// TwinCAT 3 PLC project PLC
// ProgramVersion: 3.1.4023.0
// libraries:
//   Tc2_ModbusRTU, * (Beckhoff Automation GmbH)
//   Tc2_Standard, * (Beckhoff Automation GmbH)
//   Tc2_System, * (Beckhoff Automation GmbH)
//   Tc2_Utilities, * (Beckhoff Automation GmbH)
//   Tc3_Module, * (Beckhoff Automation GmbH)
//   VisuSymbols,3.5.10.0,System
// project tree:
//   / GlobalTextList.TcGTLO, PlcTask.TcTTO, VISU_TASK.TcTTO
//   POUs/ FB_CalculateAI.TcPOU, FB_Modbus.TcPOU, FB_ModbusMaster.TcPOU, FB_ModbusSlave.TcPOU, FB_PM2200.TcPOU, FB_TDS3000.TcPOU, FB_TDS4339.TcPOU, I_ModbusSlave.TcIO (not stored), MAIN.TcPOU, U_Word2Real.TcDUT
//   VISUs/ Visualization.TcVIS, VisualizationManager.TcVMO (not stored)
// real-time tasks:
//   TASK PlcTask: cycle T#10ms, priority 20, ADS port 350
//   TASK VISU_TASK: cycle T#200000us, priority 30, ADS port 351
// I/O:
//   DEVICE Device 1 (EtherCAT) (disabled), AmsNetId 10.20.253.152.2.1
//     Term 1 (EK1200) [EK1200-5000 EtherCAT Power supply (2A E-Bus)]
//       Term 16 (EL1859) [EL1859 8Ch. Dig. Input 24V, 3ms, 8Ch. Dig. Output 24V, 0.5A]
//       Term 17 (EL1859) [EL1859 8Ch. Dig. Input 24V, 3ms, 8Ch. Dig. Output 24V, 0.5A]
//       Term 2 (EL1819) [EL1819 16Ch. Dig. Input 24V, 10µs]
//       Term 3 (EL1819) [EL1819 16Ch. Dig. Input 24V, 10µs]
//       Term 4 (EL1819) [EL1819 16Ch. Dig. Input 24V, 10µs]
//       Term 5 (EL1819) [EL1819 16Ch. Dig. Input 24V, 10µs]
//       Term 6 (EL1819) [EL1819 16Ch. Dig. Input 24V, 10µs]
//       Term 7 (EL1819) [EL1819 16Ch. Dig. Input 24V, 10µs]
//       Term 8 (EL1819) [EL1819 16Ch. Dig. Input 24V, 10µs]
//       Term 9 (EL2809) [EL2809 16Ch. Dig. Output 24V, 0.5A]
//       Term 10 (EL2809) [EL2809 16Ch. Dig. Output 24V, 0.5A]
//       Term 11 (EL3058) [EL3058 8Ch. Ana. Input 4-20mA]
//       Term 12 (EL6021) [EL6021 Interface (RS422/485)]
//       Term 30 (EL6021) [EL6021 Interface (RS422/485)]
//       Term 14 (EL9011) [EL9011 End Terminal]
//   DEVICE Device 2 (EtherCAT) (disabled), AmsNetId 192.168.56.1.3.1
//     Term 13 (EK1100) [EK1100 EtherCAT Coupler (2A E-Bus)]
//       Term 15 (EL6021) [EL6021 Interface (RS422/485)]
//   DEVICE Device 3 (COM Port)
// variable links:
//   PLC/PLC Instance <-> Device 1 (EtherCAT)/Term 1 (EK1200)/Term 10 (EL2809)
//     PlcTask Outputs/MAIN.bDO21 <-> Channel 1/Output
//     PlcTask Outputs/MAIN.bDO210 <-> Channel 10/Output
//     PlcTask Outputs/MAIN.bDO211 <-> Channel 11/Output
//     PlcTask Outputs/MAIN.bDO212 <-> Channel 12/Output
//     PlcTask Outputs/MAIN.bDO213 <-> Channel 13/Output
//     PlcTask Outputs/MAIN.bDO214 <-> Channel 14/Output
//     PlcTask Outputs/MAIN.bDO215 <-> Channel 15/Output
//     PlcTask Outputs/MAIN.bDO216 <-> Channel 16/Output
//     PlcTask Outputs/MAIN.bDO22 <-> Channel 2/Output
//     PlcTask Outputs/MAIN.bDO23 <-> Channel 3/Output
//     PlcTask Outputs/MAIN.bDO24 <-> Channel 4/Output
//     PlcTask Outputs/MAIN.bDO25 <-> Channel 5/Output
//     PlcTask Outputs/MAIN.bDO26 <-> Channel 6/Output
//     PlcTask Outputs/MAIN.bDO27 <-> Channel 7/Output
//     PlcTask Outputs/MAIN.bDO28 <-> Channel 8/Output
//     PlcTask Outputs/MAIN.bDO29 <-> Channel 9/Output
//   PLC/PLC Instance <-> Device 1 (EtherCAT)/Term 1 (EK1200)/Term 11 (EL3058)
//     PlcTask Inputs/MAIN.AI_DraftT1Case_Pressure <-> AI Standard Channel 7/Value
//     PlcTask Inputs/MAIN.AI_DraftT2Case_Voltage <-> AI Standard Channel 8/Value
//     PlcTask Inputs/MAIN.AI_Excitatiob_Current <-> AI Standard Channel 4/Value
//     PlcTask Inputs/MAIN.AI_Excitatiob_Voltage <-> AI Standard Channel 3/Value
//     PlcTask Inputs/MAIN.AI_GovernorBlOilade_Pressure <-> AI Standard Channel 2/Value
//     PlcTask Inputs/MAIN.AI_GovernorGuideVaneOil_Preesure <-> AI Standard Channel 1/Value
//     PlcTask Inputs/MAIN.AI_HeadCase_Pressure <-> AI Standard Channel 6/Value
//     PlcTask Inputs/MAIN.AI_SpiralCase_Pressure <-> AI Standard Channel 5/Value
//   PLC/PLC Instance <-> Device 1 (EtherCAT)/Term 1 (EK1200)/Term 9 (EL2809)
//     PlcTask Outputs/MAIN.bDO11 <-> Channel 1/Output
//     PlcTask Outputs/MAIN.bDO110 <-> Channel 10/Output
//     PlcTask Outputs/MAIN.bDO111 <-> Channel 11/Output
//     PlcTask Outputs/MAIN.bDO112 <-> Channel 12/Output
//     PlcTask Outputs/MAIN.bDO113 <-> Channel 13/Output
//     PlcTask Outputs/MAIN.bDO114 <-> Channel 14/Output
//     PlcTask Outputs/MAIN.bDO115 <-> Channel 15/Output
//     PlcTask Outputs/MAIN.bDO116 <-> Channel 16/Output
//     PlcTask Outputs/MAIN.bDO12 <-> Channel 2/Output
//     PlcTask Outputs/MAIN.bDO13 <-> Channel 3/Output
//     PlcTask Outputs/MAIN.bDO14 <-> Channel 4/Output
//     PlcTask Outputs/MAIN.bDO15 <-> Channel 5/Output
//     PlcTask Outputs/MAIN.bDO16 <-> Channel 6/Output
//     PlcTask Outputs/MAIN.bDO17 <-> Channel 7/Output
//     PlcTask Outputs/MAIN.bDO18 <-> Channel 8/Output
//     PlcTask Outputs/MAIN.bDO19 <-> Channel 9/Output

CONFIGURATION PLC
    RESOURCE PLC ON TwinCAT3
        TASK PlcTask(INTERVAL := T#10ms, PRIORITY := 20);
        TASK VISU_TASK(INTERVAL := T#200000us, PRIORITY := 30);
        PROGRAM MAIN WITH PlcTask : MAIN;
        PROGRAM VisuElems_Visu_Prg WITH VISU_TASK : VisuElems.Visu_Prg;
    END_RESOURCE
END_CONFIGURATION

// ---- POUs/U_Word2Real.TcDUT
TYPE U_Word2Real :
UNION
	iWord: ARRAY [0..1] OF WORD;
	rReal: REAL;
END_UNION
END_TYPE

// ---- POUs/MAIN.TcPOU
PROGRAM MAIN
VAR
	bDO11 AT %Q* :BOOL;
	bDO12 AT %Q*	:BOOL;
	bDO13 AT %Q*	:BOOL;
	bDO14 AT %Q*	:BOOL;
	bDO15 AT %Q*	:BOOL;
	bDO16 AT %Q*	:BOOL;
	bDO17 AT %Q*	:BOOL;
	bDO18 AT %Q*	:BOOL;
	bDO19 AT %Q*	:BOOL;
	bDO110 AT %Q* :BOOL;
	bDO111 AT %Q* :BOOL;
	bDO112 AT %Q* :BOOL;
	bDO113 AT %Q* :BOOL;
	bDO114 AT %Q* :BOOL;
	bDO115 AT %Q* :BOOL;
	bDO116 AT %Q* :BOOL;
		
	bDO21 AT %Q* :BOOL;
	bDO22 AT %Q*:BOOL;
	bDO23 AT %Q*:BOOL;
	bDO24 AT %Q*:BOOL;
	bDO25 AT %Q*:BOOL;
	bDO26 AT %Q*:BOOL;
	bDO27 AT %Q*:BOOL;
	bDO28 AT %Q*:BOOL;
	bDO29 AT %Q*:BOOL;
	bDO210 AT %Q* :BOOL;
	bDO211 AT %Q* :BOOL;
	bDO212 AT %Q* :BOOL;
	bDO213 AT %Q* :BOOL;
	bDO214 AT %Q* :BOOL;
	bDO215 AT %Q* :BOOL;
	bDO216 AT %Q* :BOOL;
	
	AI_GovernorGuideVaneOil_Preesure 	AT%I* :WORD;
	AI_GovernorBlOilade_Pressure 		AT%I* :WORD;
	AI_Excitatiob_Voltage 				AT%I* :WORD;
	AI_Excitatiob_Current 				AT%I* :WORD;
	AI_SpiralCase_Pressure 				AT%I* :WORD;
	AI_HeadCase_Pressure 				AT%I* :WORD;
	AI_DraftT1Case_Pressure 			AT%I* :WORD;
	AI_DraftT2Case_Voltage 				AT%I* :WORD;
	
	wGovernorGuideVaneOilPreesure 	:WORD;
	wGovernorBlOiladePressure 		:WORD;
	wExcitationVoltage 				:WORD;
	wExcitationCurrent 				:WORD;
	wSpiralCasePressure 			:WORD;
	wHeadCasePressure 				:WORD;
	wDraftT1CasePressure 			:WORD;
	wDraftT2CaseVoltage 			:WORD;
	
	lrGovernorGuideVaneOilPreesure 	:LREAL;
	lrGovernorBladeOilPressure 		:LREAL;
	lrExcitationVoltage 			:LREAL;
	lrExcitationCurrent 			:LREAL;
	lrSpiralCasePressure 			:LREAL;
	lrHeadCasePressure 				:LREAL;
	lrDraftT1CasePressure 			:LREAL;
	lrDraftT2CasePressure 			:LREAL;
	
	fbCal1	: FB_CalculateAI;
	fbCal2	: FB_CalculateAI;
	fbCal3	: FB_CalculateAI;
	fbCal4	: FB_CalculateAI;
	fbCal5	: FB_CalculateAI;
	fbCal6	: FB_CalculateAI;
	fbCal7	: FB_CalculateAI;
	fbCal8	: FB_CalculateAI;
	
	fbModbus : FB_Modbus;
END_VAR

//Assignment input
	wGovernorGuideVaneOilPreesure 	:= AI_GovernorGuideVaneOil_Preesure ;
	wGovernorBlOiladePressure 		:= AI_GovernorBlOilade_Pressure ;
	wExcitationVoltage 				:= AI_Excitatiob_Voltage;
	wExcitationCurrent 				:= AI_Excitatiob_Current;
	wSpiralCasePressure 			:= AI_SpiralCase_Pressure;
	wHeadCasePressure 				:= AI_HeadCase_Pressure ;
	wDraftT1CasePressure 			:= AI_DraftT1Case_Pressure ;
	wDraftT2CaseVoltage 			:= AI_DraftT2Case_Voltage ;
	
//Calculate input
	//Chanel 1 data
		fbCal1.MaxEngIn := LREAL_TO_WORD(6);
		fbCal1.MinEngIn	:= LREAL_TO_WORD(0);
		fbCal1.RawIn := wGovernorGuideVaneOilPreesure;
		fbCal1.Description:= 'MPa';
		
	//Chanel 2 data
		fbCal2.MaxEngIn := LREAL_TO_WORD(25);
		fbCal2.MinEngIn	:= LREAL_TO_WORD(0);
		fbCal2.RawIn := wGovernorBlOiladePressure ;
		fbCal2.Description:= 'MPa';
	
	//Chanel 3 data
		fbCal3.MaxEngIn := LREAL_TO_WORD(300);
		fbCal3.MinEngIn	:= LREAL_TO_WORD(0);
		fbCal3.RawIn := wExcitationVoltage;
		fbCal3.Description:= 'V';
		
	//Chanel 4 data
		fbCal4.MaxEngIn := LREAL_TO_WORD(500);
		fbCal4.MinEngIn	:= LREAL_TO_WORD(0);
		fbCal4.RawIn := wExcitationCurrent ;
		fbCal4.Description:= 'A';
		
	//Chanel 5 data
		fbCal5.MaxEngIn := LREAL_TO_WORD(0.4*1000);
		fbCal5.MinEngIn	:= LREAL_TO_WORD(0*1000);
		fbCal5.RawIn := wSpiralCasePressure;
		fbCal5.Description:= 'MPa';
		
	//Chanel 6 data
		fbCal6.MaxEngIn := LREAL_TO_WORD(0.3*1000);
		fbCal6.MinEngIn	:= LREAL_TO_WORD(-0.1*1000);
		fbCal6.RawIn := wHeadCasePressure;
		fbCal6.Description:= 'MPa';
		
	//Chanel 7 data
		fbCal7.MaxEngIn := LREAL_TO_WORD(0.3*1000);
		fbCal7.MinEngIn	:= LREAL_TO_WORD(-0.1*1000);
		fbCal7.RawIn := wDraftT1CasePressure;
		fbCal7.Description:= 'MPa';
		
	//Chanel 8 data
		fbCal8.MaxEngIn := LREAL_TO_WORD(0.3*1000);
		fbCal8.MinEngIn	:= LREAL_TO_WORD(-0.1*1000);
		fbCal8.RawIn := wDraftT2CaseVoltage;
		fbCal8.Description:= 'MPa';

// Call FB
	fbCal1();
	fbCal2();
	fbCal3();
	fbCal4();
	fbCal5();
	fbCal6();
	fbCal7();
	fbCal8();
		
//Calculate output
	//Chanel 1 output
		lrGovernorGuideVaneOilPreesure := fbCal1.CalVal;
		
	//Chanel 2 output
		lrGovernorBladeOilPressure := fbCal2.CalVal;
		
	//Chanel 3 output
		lrExcitationVoltage := fbCal3.CalVal;
		
	//Chanel 4 output
		lrExcitationCurrent := fbCal4.CalVal;
		
	//Chanel 5 output
		lrSpiralCasePressure := fbCal5.CalVal/1000;
		
	//Chanel 6 output
		lrHeadCasePressure := fbCal6.CalVal/1000;
		
	//Chanel 7 output
		lrDraftT1CasePressure := fbCal7.CalVal/1000;
		
	//Chanel 8 output
		lrDraftT2CasePressure := fbCal8.CalVal/1000;

fbModbus();

END_PROGRAM

// ---- POUs/FB_CalculateAI.TcPOU
FUNCTION_BLOCK FB_CalculateAI
VAR_INPUT
END_VAR
VAR_OUTPUT
END_VAR
VAR
	wMinRawIn		: WORD := 0;
	wMaxRawIn		: WORD := 32767;
	wRawIn			: WORD;
	wMinEngIn		: WORD;
	wMaxEngIn		: WORD;
	lrCalVal			: lreal;
	sDescription 	: STRING;
	lrRes			: LREAL;
	
END_VAR

lrRes := WORD_TO_LREAL(wRawIn)/WORD_TO_LREAL(wMaxRawIn);
lrCalVal:= word_to_lreal(wMaxEngIn) * lrRes;

PROPERTY CalVal : LREAL
GET
Calval := lrCalVal;
END_GET
SET
lrCalVal := Calval;
END_SET
END_PROPERTY

PROPERTY Description : STRING
SET
sDescription := Description;
END_SET
END_PROPERTY

PROPERTY MaxEngIn : WORD
SET
wMaxEngIn := MaxEngIn;
END_SET
END_PROPERTY

PROPERTY MinEngIn : WORD
SET
wMinEngIn := MinEngIn;
END_SET
END_PROPERTY

PROPERTY RawIn : WORD
SET
wRawIn := RawIn;
END_SET
END_PROPERTY

END_FUNCTION_BLOCK

// ---- POUs/FB_Modbus.TcPOU
FUNCTION_BLOCK FB_Modbus
VAR_INPUT
END_VAR
VAR_OUTPUT
END_VAR
VAR
	fbModbusMaster1 :		FB_ModbusMaster;
	fbModbusMaster2 :		FB_ModbusMaster;
	fbModbusSlave	:		FB_PM2200;
	fbModbusSlave1	: 		FB_TDS3000;
	fbModbusSlave2	: 		FB_TDS3000;
	fbModbusSlave3	: 		FB_TDS3000;
	istep			:		UINT;
	bStart			:		BOOL;
	
	arrData			:		ARRAY [0..255] OF BYTE := [1,3,12,16#00,16#01,16#01,16#02,16#03,16#01,16#01,16#01,16#01,16#01,16#01,16#01,3,5] ;
END_VAR

CASE istep OF
	0: //Trigger
		IF bStart THEN
			bStart := FALSE;
			istep := 10;
		END_IF
		
	10: //Init
		fbModbusSlave.UnitID := 1;
		fbModbusSlave.FirstCycle();
		
		fbModbusSlave1.UnitID := 1;
		fbModbusSlave1.FirstCycle();
		fbModbusSlave2.UnitID := 2;
		fbModbusSlave2.FirstCycle();
		fbModbusSlave3.UnitID := 3;
		fbModbusSlave3.FirstCycle();
		
		fbModbusMaster1.FirstCycle();
		fbModbusMaster1.Init();
		fbModbusMaster1.RegisterSlave(fbModbusSlave);
//		fbModbusMaster.RegisterSlave(fbModbusTemp);
		fbModbusMaster1.Timeout := 1000;
		
		fbModbusMaster2.FirstCycle();
		fbModbusMaster2.Init();
		fbModbusMaster2.RegisterSlave(fbModbusSlave1);
		fbModbusMaster2.RegisterSlave(fbModbusSlave2);
		fbModbusMaster2.RegisterSlave(fbModbusSlave3);
		fbModbusMaster2.Timeout := 1000;
		
		istep := 20;
		
	20: //Running
		IF fbModbusMaster1.Run()AND fbModbusMaster2.Run() THEN
			istep := 30;
		END_IF
		
	30: //Stopped
		
END_CASE

fbModbusMaster1();
fbModbusMaster2();

fbModbusSlave.Convert(0, ADR(arrData));

END_FUNCTION_BLOCK

// ---- POUs/FB_ModbusMaster.TcPOU
FUNCTION_BLOCK FB_ModbusMaster //IMPLEMENTS I_UniversalUnit
VAR
	sName			:		STRING;
	bInitialized	:		BOOL;
	iScantime		:		UINT;
	iTimeout		:		UINT;
	//iErrorID		:		UDINT;
	iErrorID		:		MODBUS_ERRORS;
	
	bBusy			: 		BOOL;
	bError			:		BOOL;
	
	iStepInit		:		INT;
	iStepGeneral	: 		INT;
	iStepRunning	:		INT;
	bFirstCycle		:		BOOL;
	
	bRun			:		BOOL;
	bStop			: 		BOOL;
	
	fbModbusMaster	: 		ModbusRtuMaster_PcCOM;
//	fbModbusMaster : 		ModbusRtuMaster_KL6x22B;
	ipModbusSlave	:		ARRAY [1..247] OF I_ModbusSlave;
	iAmountSlave	: 		UINT;
	
	iLoopSlave		:		UINT	:= 1;
	iLoopAdr		:		UINT;
	iQuantity 		: 		POINTER TO WORD;
	iMBAddr 		: 		POINTER TO WORD;
    arrData			: 		ARRAY [0..255] OF BYTE;
	
	bDelayState		:		BOOL;
	
END_VAR

IF bFirstCycle THEN
	bFirstCycle := FALSE;
END_IF
		
StateMachine();

bRun := FALSE;
bStop := FALSE;

bInitialized := iStepGeneral >= 20;

bError S= fbModbusMaster.Error AND iStepGeneral = 30 and iStepRunning = 60;
bError R= NOT fbModbusMaster.Error AND iStepGeneral = 30 AND iStepRunning = 60;
IF iStepGeneral = 30 AND iStepRunning = 60 THEN
	iErrorID := fbModbusMaster.ErrorId;
END_IF

bBusy := fbModbusMaster.BUSY AND iStepGeneral = 30;

//	// error	
//		fbAxisError.Description := FUN_MergeStrings5(sMotorName, ' axis error number: ', UDINT_TO_STRING(iErrorID), '', '');
//		fbAxisError.Set(bError);

METHOD Abort : BOOL
END_METHOD

PROPERTY AnyError : BOOL
GET
AnyError 	:= bError;
END_GET
END_PROPERTY

PROPERTY Busy : BOOL
GET
Busy := bBusy;
END_GET
END_PROPERTY

PROPERTY ErrorID : UDINT
GET
ErrorID := iErrorID;
END_GET
END_PROPERTY

METHOD FirstCycle : BOOL
VAR_INPUT
//	ipAlarmController	: I_AlarmController;
//	ipHMIController	: I_HMIController;
END_VAR
END_METHOD

METHOD Init : BOOL
IF iStepGeneral = 0 THEN
	iStepGeneral := 10;
END_IF

//Method output
	Init := (iStepGeneral >= 20);
END_METHOD

PROPERTY Initialized : BOOL
GET
Initialized := bInitialized;
END_GET
END_PROPERTY

PROPERTY Name : STRING
GET
Name := sName;
END_GET
SET
sName := Name;
END_SET
END_PROPERTY

PROPERTY ReadData : ARRAY [0..255] OF BYTE
GET
ReadData := arrData;
END_GET
END_PROPERTY

PROPERTY ReadDataSize : uint
GET
ReadDataSize := INT_TO_UINT(SIZEOF(arrData));
END_GET
END_PROPERTY

METHOD RegisterSlave : BOOL
VAR_INPUT
	ModbusSlave		:		I_ModbusSlave;
END_VAR
VAR
	iLoop	:	UINT;
	bExists	:	BOOL;
END_VAR
FOR iLoop := 1 TO iAmountSlave DO
	IF ipModbusSlave[iLoop] = ModbusSlave THEN
		bExists := TRUE;
		iLoop := iAmountSlave;
	END_IF
END_FOR 
IF NOT bExists THEN
	iAmountSlave := iAmountSlave + 1;
	ipModbusSlave[iAmountSlave] := ModbusSlave;
END_IF
END_METHOD

METHOD Reset : BOOL
bError := FALSE;
iErrorID := 0;
bError := FALSE;
iStepInit		:= 0;
iStepGeneral	:= 0;
iStepRunning	:= 0;

iLoopSlave		:= 1;
iLoopAdr		:= 0;

fbModbusMaster.Execute := FALSE;

Reset := TRUE;
END_METHOD

METHOD Run : BOOL
IF (iStepGeneral = 20) THEN
	iStepGeneral := 30;
END_IF

bRun := TRUE;
Run := (iStepGeneral >= 30) AND (iStepGeneral < 200);
END_METHOD

PROPERTY ScanTime : UINT
GET
ScanTime := iScantime;
END_GET
SET
iScantime := ScanTime;
END_SET
END_PROPERTY

METHOD StateInit : BOOL (*Unit is performing initialization*)
IF NOT bError THEN
	iStepGeneral := 20;
END_IF
END_METHOD

METHOD StateMachine : BOOL (*State machine of unit*)
//State machine						   
	CASE iStepGeneral OF
		0:  //Uninitialized
			StateUninitialized();
	
		10: //Initializing
			StateInit();
	
		20: //Ready
			StateReady();
		
		30: //Running
			StateRunning();
						
		200: //stop
			StateStopping();
			
		210: //stop done
			StateStoppingDone();
	END_CASE
END_METHOD

METHOD StateReady : BOOL (* Unit is initialized*)
END_METHOD

METHOD StateRunning : BOOL (* Unit is uninitialized*)
VAR 
END_VAR
CASE iStepRunning OF
	0: // Trigger
		IF iAmountSlave > 0 THEN
			iStepRunning := 10;
		ELSE
			iStepRunning := 50;
		END_IF
		
	10: // Set parameters
		IF iLoopSlave <= iAmountSlave THEN
			IF  iLoopAdr <= ipModbusSlave[iLoopSlave].NumAddRegion - 1 THEN
				iQuantity := (ipModbusSlave[iLoopSlave].Address + (iLoopAdr*2+1)*SIZEOF(WORD));
				iMBAddr := (ipModbusSlave[iLoopSlave].Address + (iLoopAdr*2)*SIZEOF(WORD));
				
				fbModbusMaster.UnitID 	:=		ipModbusSlave[iLoopSlave].UnitID;
				fbModbusMaster.Quantity	:=		iQuantity^;
				fbModbusMaster.MBAddr	:=		iMBAddr^;
				fbModbusMaster.cbLength	:= 		SIZEOF(arrData);
				fbModbusMaster.pMemoryAddr	:= 	ADR(arrData);
				fbModbusMaster.Timeout	:= 		UINT_TO_TIME(iTimeout);
				
				iLoopAdr := iLoopAdr + 1;
				iStepRunning := 20;
			ELSE
				iLoopAdr := 0;
				iLoopSlave := iLoopSlave + 1;
				iStepRunning := 60;
				bDelayState := NOT bDelayState;
			END_IF
		ELSE
			iLoopSlave := 1;
			iStepRunning := 60;
			bDelayState := NOT bDelayState;
		END_IF
		
	20: // Send request
		IF NOT fbModbusMaster.BUSY THEN
			iStepRunning := 30;
		END_IF
	
	30: // Wait ack request
		IF fbModbusMaster.BUSY THEN
			iStepRunning := 40;
		END_IF
		
	40: // Wait respond
		IF NOT fbModbusMaster.BUSY THEN
			iStepRunning := 50;
		END_IF
		
	50: // Convert raw data
		IF iLoopSlave <= iAmountSlave THEN
			ipModbusSlave[iLoopSlave].Convert(iLoopAdr, ADR(arrData));
		END_IF
		bDelayState := NOT bDelayState;
		iStepRunning := 60;

	60: // Return, done
		IF NOT bDelayState THEN
			iStepRunning := 0;
		END_IF
		bDelayState := NOT bDelayState;
		
END_CASE

IF (iStepRunning >= 20) AND (iStepRunning <= 40) THEN
	fbModbusMaster.ReadRegs();
END_IF
fbModbusMaster.Execute := iStepRunning >= 20 AND iStepRunning <= 30;


//bTest S= iStepRunning > 
//tonTest(IN :=
END_METHOD

METHOD StateStopping : BOOL (* Unit is uninitialized*)
iStepGeneral	:= 0;
iStepRunning	:= 210;

iLoopSlave		:= 1;
iLoopAdr		:= 0;

fbModbusMaster.Execute := FALSE;
END_METHOD

METHOD StateStoppingDone : BOOL (* Unit is uninitialized*)
IF NOT bStop THEN
	iStepGeneral := 20;
END_IF
END_METHOD

METHOD StateUninitialized : BOOL (* Unit is uninitialized*)
END_METHOD

METHOD Stop : BOOL
IF iStepGeneral >= 30 AND iStepGeneral < 200 THEN
	iStepGeneral := 200;
END_IF
bStop := TRUE;

Stop := (iStepGeneral = 210);
END_METHOD

PROPERTY Timeout : UINT
GET
Timeout := iTimeout;
END_GET
SET
iTimeout := Timeout;
END_SET
END_PROPERTY

END_FUNCTION_BLOCK

// ---- POUs/FB_PM2200.TcPOU
FUNCTION_BLOCK FB_PM2200 EXTENDS FB_ModbusSlave
VAR
	// Current
		rCurrentA		:		REAL;
		rCurrentB		:		REAL;
		rCurrentC		:		REAL;
		rCurrentN		:		REAL;
		rCurrentG		:		REAL;
		rCurrentAvg		:		REAL;
	
	// Voltage
		rVoltageAB		:		REAL;
		rVoltageBC		:		REAL;
		rVoltageCA		:		REAL;
		rVoltageLLAvg	:		REAL;
		rVoltageAN		:		REAL;
		rVoltageBN		:		REAL;
		rVoltageCN		:		REAL;
		rVoltageLNAvg	:		REAL;
		
	// Power
		rActivePowerA	:		REAL;
		rActivePowerB	:		REAL;
		rActivePowerC	:		REAL;
		rActivePowerTotal	:	REAL;
		rReactivePowerA	:		REAL;
		rReactivePowerB	:		REAL;
		rReactivePowerC	:		REAL;
		rReactivePowerTotal	:	REAL;
		rApparentPowerA	:		REAL;
		rApparentPowerB	:		REAL;
		rApparentPowerC	:		REAL;
		rApparentPowerTotal	:	REAL;
		
	// Power factor
		rPowerFactorA	:		REAL;
		rPowerFactorB	:		REAL;
		rPowerFactorC	:		REAL;
		rPowerFactorTotal	:	REAL;
		rDisPowerFactorA	:	REAL;
		rDisPowerFactorB	:	REAL;
		rDisPowerFactorC	:	REAL;
		rDisPowerFactorTotal:	REAL;

	// Frequency
		rFrequency		: 		REAL;
		
END_VAR

PROPERTY ActivePowerA : REAL
GET
ActivePowerA := rActivePowerA;
END_GET
END_PROPERTY

PROPERTY ActivePowerB : REAL
GET
ActivePowerB := rActivePowerB;
END_GET
END_PROPERTY

PROPERTY ActivePowerC : REAL
GET
ActivePowerC := rActivePowerC;
END_GET
END_PROPERTY

PROPERTY ActivePowerTotal : REAL
GET
ActivePowerTotal := rActivePowerTotal;
END_GET
END_PROPERTY

PROPERTY ApparentPowerA : REAL
GET
ApparentPowerA := rApparentPowerA;
END_GET
END_PROPERTY

PROPERTY ApparentPowerB : REAL
GET
ApparentPowerB := rApparentPowerB;
END_GET
END_PROPERTY

PROPERTY ApparentPowerC : REAL
GET
ApparentPowerC := rApparentPowerC;
END_GET
END_PROPERTY

PROPERTY ApparentPowerTotal : REAL
GET
ApparentPowerTotal := rApparentPowerTotal;
END_GET
END_PROPERTY

METHOD Convert : BOOL
VAR_INPUT
	iRegionNo	:	INT;
	pReadData	:	POINTER TO BYTE;
END_VAR
VAR
	iTempDataHi	: 	BYTE;
	iTempDataLo	:	BYTE;
	iLoop		: 	INT;
	bHiByte		:	BOOL := TRUE;
	arrTempData	:	ARRAY [0..3] OF U_Word2Real;
END_VAR
FOR iLoop := 0 TO 3 DO
	arrTempData[iLoop].iWord[1] := SHL(BYTE_TO_WORD(pReadData[iLoop*4+3]), 8);
	arrTempData[iLoop].iWord[1] := arrTempData[iLoop].iWord[1] + BYTE_TO_WORD(pReadData[iLoop*4+3+1]);
	arrTempData[iLoop].iWord[0] := SHL(BYTE_TO_WORD(pReadData[iLoop*4+3+2]), 8);
	arrTempData[iLoop].iWord[0] := arrTempData[iLoop].iWord[0] + BYTE_TO_WORD(pReadData[iLoop*4+3+3]);
	IF bSwap THEN
		arrTempData[iLoop].iWord[0] := ROL(arrTempData[iLoop].iWord[0], 8);
		arrTempData[iLoop].iWord[1] := ROL(arrTempData[iLoop].iWord[1], 8);
	END_IF
END_FOR

CASE iRegionNo OF
	0: 
		rCurrentA := arrTempData[0].rReal;
		rCurrentB := arrTempData[1].rReal;
		rCurrentC := arrTempData[2].rReal;
		rCurrentN := arrTempData[3].rReal;

	1:
		rCurrentG := arrTempData[0].rReal;
		rCurrentAvg := arrTempData[1].rReal;

		
	2: 
		rVoltageAB := arrTempData[0].rReal;
		rVoltageBC := arrTempData[1].rReal;
		rVoltageCA := arrTempData[2].rReal;
		rVoltageLLAvg := arrTempData[3].rReal;
		
	3:
		rVoltageAN := arrTempData[0].rReal;
		rVoltageBN := arrTempData[1].rReal;
		rVoltageCN := arrTempData[2].rReal;
		rVoltageLNAvg := arrTempData[3].rReal;

	4: 
		rActivePowerA := arrTempData[0].rReal;
		rActivePowerB := arrTempData[1].rReal;
		rActivePowerC := arrTempData[2].rReal;
		rActivePowerTotal := arrTempData[3].rReal;
		
	5:
		rReactivePowerA := arrTempData[0].rReal;
		rReactivePowerB := arrTempData[1].rReal;
		rReactivePowerC := arrTempData[2].rReal;
		rReactivePowerTotal := arrTempData[3].rReal;
		
	6: 
		rApparentPowerA := arrTempData[0].rReal;
		rApparentPowerB := arrTempData[1].rReal;
		rApparentPowerC := arrTempData[2].rReal;
		rApparentPowerTotal := arrTempData[3].rReal;
		
	7:
		rPowerFactorA := arrTempData[0].rReal;
		rPowerFactorB := arrTempData[1].rReal;
		rPowerFactorC := arrTempData[2].rReal;
		rPowerFactorTotal := arrTempData[3].rReal;

	8:
		rDisPowerFactorA := arrTempData[0].rReal;
		rDisPowerFactorB := arrTempData[1].rReal;
		rDisPowerFactorC := arrTempData[2].rReal;
		rDisPowerFactorTotal := arrTempData[3].rReal;
		
	9:	
		rFrequency := arrTempData[0].rReal;

END_CASE
END_METHOD

PROPERTY CurrentA : REAL
GET
CurrentA := rCurrentA;
END_GET
END_PROPERTY

PROPERTY CurrentAvg : REAL
GET
CurrentAvg := rCurrentAvg;
END_GET
END_PROPERTY

PROPERTY CurrentB : REAL
GET
CurrentB := rCurrentB;
END_GET
END_PROPERTY

PROPERTY CurrentC : REAL
GET
CurrentC := rCurrentC;
END_GET
END_PROPERTY

PROPERTY CurrentG : REAL
GET
CurrentG := rCurrentG;
END_GET
END_PROPERTY

PROPERTY CurrentN : REAL
GET
CurrentN := rCurrentN;
END_GET
END_PROPERTY

METHOD FirstCycle : BOOL
VAR_INPUT
END_VAR
arrAddress[0][0] := 2999;			// Current A & B & C & N
arrAddress[0][1] := 16;
arrAddress[1][0] := 3007;			// Current G & Avg
arrAddress[1][1] := 8;

arrAddress[2][0] := 3019;			// Voltage AB, BC, CA, LL Avg
arrAddress[2][1] := 16;		
arrAddress[3][0] := 3027;			// Voltage AN, BN, CN, LN Avg
arrAddress[3][1] := 16;		
		
arrAddress[4][0] := 3053;			// Active Power 
arrAddress[4][1] := 16;				
arrAddress[5][0] := 3061;			// Reactive Power
arrAddress[5][1] := 16;			
arrAddress[6][0] := 3069;			// Apparent Power
arrAddress[6][1] := 16;				

arrAddress[7][0] := 3077;			// Power factor
arrAddress[7][1] := 16;		
arrAddress[8][0] := 3085;			// Displacement Power factor
arrAddress[8][1] := 16;		
		
arrAddress[9][0] := 3109;			// Frequency
arrAddress[9][1] := 4;				

iNumAddRegion := 10;

bSwap := FALSE;
END_METHOD

PROPERTY Frequency : REAL
GET
Frequency := rFrequency;
END_GET
END_PROPERTY

PROPERTY PowerFactorA : REAL
GET
PowerFactorA := rPowerFactorA;
END_GET
END_PROPERTY

PROPERTY PowerFactorB : REAL
GET
PowerFactorB := rPowerFactorB;
END_GET
END_PROPERTY

PROPERTY PowerFactorC : REAL
GET
PowerFactorC := rPowerFactorC;
END_GET
END_PROPERTY

PROPERTY PowerFactorTotal : REAL
GET
PowerFactorTotal := rPowerFactorTotal;
END_GET
END_PROPERTY

PROPERTY ReActivePowerA : REAL
GET
ReActivePowerA := rReactivePowerA;
END_GET
END_PROPERTY

PROPERTY ReActivePowerB : REAL
GET
ReActivePowerB := rReactivePowerB;
END_GET
END_PROPERTY

PROPERTY ReActivePowerC : REAL
GET
ReActivePowerC := rReactivePowerC;
END_GET
END_PROPERTY

PROPERTY ReActivePowerTotal : REAL
GET
ReActivePowerTotal := rReactivePowerTotal;
END_GET
END_PROPERTY

PROPERTY VoltageAB : REAL
GET
VoltageAB := rVoltageAB;
END_GET
END_PROPERTY

PROPERTY VoltageAN : REAL
GET
VoltageAN := rVoltageAN;
END_GET
END_PROPERTY

PROPERTY VoltageBC : REAL
GET
VoltageBC := rVoltageBC;
END_GET
END_PROPERTY

PROPERTY VoltageBN : REAL
GET
VoltageBN := rVoltageBN;
END_GET
END_PROPERTY

PROPERTY VoltageCA : REAL
GET
VoltageCA := rVoltageCA;
END_GET
END_PROPERTY

PROPERTY VoltageCN : REAL
GET
VoltageCN := rVoltageCN;
END_GET
END_PROPERTY

PROPERTY VoltageLLAvg : REAL
GET
VoltageLLAvg := rVoltageLLAvg;
END_GET
END_PROPERTY

PROPERTY VoltageLNAvg : REAL
GET
VoltageLNAvg := rVoltageLNAvg;
END_GET
END_PROPERTY

END_FUNCTION_BLOCK

// ---- POUs/FB_ModbusSlave.TcPOU
FUNCTION_BLOCK FB_ModbusSlave IMPLEMENTS I_ModbusSlave
VAR
	iUnitID			: 		BYTE;
	arrAddress		:		ARRAY [0..50] OF ARRAY [0..1] OF WORD;
	iNumAddRegion	:		UINT;
	bSwap			:		BOOL;
	
	sName			:		STRING;

END_VAR

PROPERTY Address : POINTER TO WORD
GET
Address := ADR(arrAddress);
END_GET
END_PROPERTY

METHOD Convert : BOOL
VAR_INPUT
	iRegionNo	:	INT;
	pReadData	:	POINTER TO BYTE;
END_VAR
END_METHOD

METHOD FirstCycle : BOOL
VAR_INPUT
END_VAR
END_METHOD

PROPERTY Name : STRING
GET
Name := sName;
END_GET
SET
sName := Name;
END_SET
END_PROPERTY

PROPERTY NumAddRegion : UINT
GET
NumAddRegion := iNumAddRegion;
END_GET
END_PROPERTY

PROPERTY UnitID : BYTE
GET
UnitID := iUnitID;
END_GET
SET
iUnitID := UnitID;
END_SET
END_PROPERTY

END_FUNCTION_BLOCK

// ---- POUs/FB_TDS3000.TcPOU
FUNCTION_BLOCK FB_TDS3000 EXTENDS FB_ModbusSlave
VAR
	arrConditionData	:	ARRAY [0..63] OF WORD;
	arrUp_LoLimit		:	ARRAY [0..63] OF WORD;
	arrUpUp_UpLimit		:	ARRAY [0..63] OF WORD;
END_VAR

PROPERTY ConditionData : ARRAY [0..63] OF WORD
GET
ConditionData := arrConditionData;
END_GET
END_PROPERTY

METHOD Convert : BOOL
VAR_INPUT
	iRegionNo	:	INT;
	pReadData	:	POINTER TO BYTE;
END_VAR
VAR
	pTempData	: 	POINTER TO BYTE;
	iTempData	: 	BYTE;
	iLoop		: 	INT;
	bHiByte		:	BOOL := TRUE;
	iLoopStart	:	INT;
	iLoopEnd	:	INT;
END_VAR
CASE iRegionNo OF
	0: 
		iLoopStart := 0;
		iLoopEnd := 15;
	
	1:
		iLoopStart := 16;
		iLoopEnd := 31;
		
	2: 
		iLoopStart := 32;
		iLoopEnd := 47;
		
	3: 
		iLoopStart := 48;
		iLoopEnd := 63;
		
END_CASE

FOR iLoop := iLoopStart TO iLoopEnd DO
	pTempData := (pReadData + iLoop);
	iTempData := pTempData^;
	
	IF bHiByte THEN
		arrConditionData[iLoop/2] := SHL(BYTE_TO_WORD(iTempData), 8);
	ELSE 
		arrConditionData[iLoop/2] := arrConditionData[iLoop/2] + BYTE_TO_WORD(iTempData);
		IF bSwap THEN
			arrConditionData[iLoop/2] := ROL(arrConditionData[iLoop/2], 8);
		END_IF
	END_IF
	bHiByte := NOT bHiByte;
END_FOR
END_METHOD

METHOD FirstCycle : BOOL
VAR_INPUT
END_VAR
arrAddress[0][0] := 16#0000;
arrAddress[0][1] := 16;
arrAddress[1][0] := 16#0008;
arrAddress[1][1] := 16;
arrAddress[2][0] := 16#0010;
arrAddress[2][1] := 16;
arrAddress[3][0] := 16#0018;
arrAddress[3][1] := 16;

iNumAddRegion := 4;

bSwap := FALSE;
END_METHOD

PROPERTY Up_LoLimit : ARRAY [0..63] OF WORD
GET
Up_LoLimit := arrUp_LoLimit;
END_GET
END_PROPERTY

PROPERTY UpUp_UpLimit : ARRAY [0..63] OF WORD
GET
UpUp_UpLimit := arrUpUp_UpLimit;
END_GET
END_PROPERTY

END_FUNCTION_BLOCK

// ---- POUs/FB_TDS4339.TcPOU
FUNCTION_BLOCK FB_TDS4339 EXTENDS FB_ModbusSlave
VAR
	rFrequency		:	REAL;
	iSpeed			:	INT;
	rPercentSpeed	:	REAL;
	rMaxFrequency	:	REAL;
	iMaxSpeed		:	INT;
	rMaxPercSpeed	:	REAL;
	rCrawlingSpeed	:	REAL;
END_VAR

METHOD Convert : BOOL
VAR_INPUT
	iRegionNo	:	INT;
	pReadData	:	POINTER TO BYTE;
END_VAR
VAR
	pTempData	: 	POINTER TO BYTE;
	iTempData	: 	BYTE;
	iLoop		: 	INT;
	bHiByte		:	BOOL := TRUE;
	arrTempData	:	ARRAY [0..6] OF WORD;
END_VAR
FOR iLoop := 0 TO 15 DO
	pTempData := (pReadData + iLoop);
	iTempData := pTempData^;
	
	IF bHiByte THEN
		arrTempData[iLoop/2] := SHL(BYTE_TO_WORD(iTempData), 8);
	ELSE 
		arrTempData[iLoop/2] := arrTempData[iLoop/2] + BYTE_TO_WORD(iTempData);
		IF bSwap THEN
			arrTempData[iLoop/2] := ROL(arrTempData[iLoop/2], 8);
		END_IF
	END_IF
	bHiByte := NOT bHiByte;
END_FOR

rFrequency := WORD_TO_REAL(arrTempData[0])/100;
iSpeed := WORD_TO_INT(arrTempData[1]);
rPercentSpeed := WORD_TO_REAL(arrTempData[2])/10;
rMaxFrequency := WORD_TO_REAL(arrTempData[3])/100;
iMaxSpeed := WORD_TO_INT(arrTempData[4]);
rMaxPercSpeed := WORD_TO_REAL(arrTempData[5])/10;
rCrawlingSpeed := WORD_TO_REAL(arrTempData[6])/100;
END_METHOD

PROPERTY CrawlingSpeed : REAL
GET
CrawlingSpeed := rCrawlingSpeed;
END_GET
END_PROPERTY

METHOD FirstCycle : BOOL
VAR_INPUT
END_VAR
arrAddress[0][0] := 16#0000;
arrAddress[0][1] := 14;

iNumAddRegion := 1;

bSwap := FALSE;
END_METHOD

PROPERTY Frequency : REAL
GET
Frequency := rFrequency;
END_GET
END_PROPERTY

PROPERTY MaxFrequency : REAL
GET
MaxFrequency := rMaxFrequency;
END_GET
END_PROPERTY

PROPERTY MaxPercentSpeed : REAL
GET
MaxPercentSpeed := rMaxPercSpeed;
END_GET
END_PROPERTY

PROPERTY MaxSpeed : INT
GET
MaxSpeed := iMaxSpeed;
END_GET
END_PROPERTY

PROPERTY PercentSpeed : REAL
GET
PercentSpeed := rPercentSpeed;
END_GET
END_PROPERTY

PROPERTY Speed : INT
GET
Speed := iSpeed;
END_GET
END_PROPERTY

END_FUNCTION_BLOCK

// ---- GlobalTextList.TcGTLO
TEXTLIST GlobalTextList
  975 = '%1.4w'
  647 = '%2.4f'
  24 = '%2.4lr'
  198 = '%2.8f'
  411 = '%5d'
  131 = '%5w'
  582 = '%s'
  795 = 'Analog 1'
  175 = 'Analog 2'
  702 = 'Analog 3'
  462 = 'Analog 4'
  289 = 'Analog 5'
  290 = 'Analog 6'
  960 = 'Analog 7'
  755 = 'Analog 8'
  512 = 'Current'
  412 = 'Current value'
  29 = 'DI 1'
  661 = 'DI 2'
  652 = 'DI 3'
  630 = 'DI 4'
  15 = 'DI 5'
  577 = 'DO 1'
  75 = 'DO 10'
  463 = 'DO 11'
  394 = 'DO 12'
  587 = 'DO 13'
  516 = 'DO 14'
  949 = 'DO 15'
  524 = 'DO 16'
  11 = 'DO 2'
  483 = 'DO 3'
  932 = 'DO 4'
  923 = 'DO 5'
  324 = 'DO 6'
  120 = 'DO 7'
  637 = 'DO 8'
  695 = 'DO 9'
  313 = 'DO15'
  109 = 'Max'
  144 = 'Min'
  969 = 'Raw value'
END_TEXTLIST

// ---- VISUs/Visualization.TcVIS
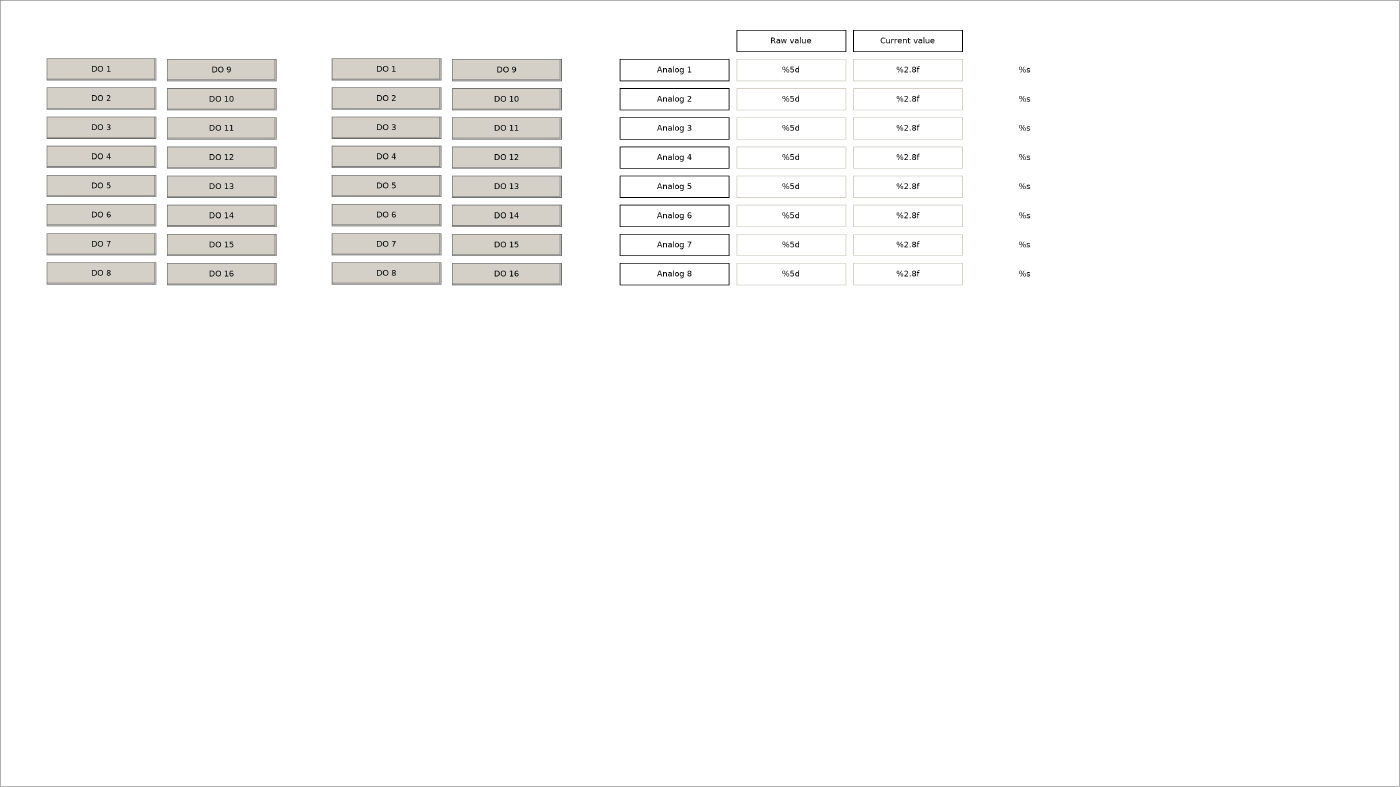
VISUALIZATION Visualization  // 1920x1080
    Button (64,80 150x30), "DO 1", colour toggle: MAIN.bDO11
        toggle MAIN.bDO11
    Button (64,120 150x30), "DO 2", colour toggle: MAIN.bDO12
        toggle MAIN.bDO12
    Button (64,160 150x30), "DO 3", colour toggle: MAIN.bDO13
        toggle MAIN.bDO13
    Button (64,200 150x30), "DO 4", colour toggle: MAIN.bDO14
        toggle MAIN.bDO14
    Button (64,240 150x30), "DO 5", colour toggle: MAIN.bDO15
        toggle MAIN.bDO15
    Button (64,280 150x30), "DO 6", colour toggle: MAIN.bDO16
        toggle MAIN.bDO16
    Button (64,320 150x30), "DO 7", colour toggle: MAIN.bDO17
        toggle MAIN.bDO17
    Button (64,360 150x30), "DO 8", colour toggle: MAIN.bDO18
        toggle MAIN.bDO18
    Button (229,81 150x30), "DO 9", colour toggle: MAIN.bDO19
        toggle MAIN.bDO19
    Button (229,121 150x30), "DO 10", colour toggle: MAIN.bDO110
        toggle MAIN.bDO110
    Button (229,161 150x30), "DO 11", colour toggle: MAIN.bDO111
        toggle MAIN.bDO111
    Button (229,201 150x30), "DO 12", colour toggle: MAIN.bDO112
        toggle MAIN.bDO112
    Button (229,241 150x30), "DO 13", colour toggle: MAIN.bDO113
        toggle MAIN.bDO113
    Button (229,281 150x30), "DO 14", colour toggle: MAIN.bDO114
        toggle MAIN.bDO114
    Button (229,321 150x30), "DO 15", colour toggle: MAIN.bDO115
        toggle MAIN.bDO115
    Button (229,361 150x30), "DO 16", colour toggle: MAIN.bDO116
        toggle MAIN.bDO116
    Button (455,80 150x30), "DO 1", colour toggle: MAIN.bDO21
        toggle MAIN.bDO21
    Button (455,120 150x30), "DO 2", colour toggle: MAIN.bDO22
        toggle MAIN.bDO22
    Button (455,160 150x30), "DO 3", colour toggle: MAIN.bDO23
        toggle MAIN.bDO23
    Button (455,200 150x30), "DO 4", colour toggle: MAIN.bDO24
        toggle MAIN.bDO24
    Button (455,240 150x30), "DO 5", colour toggle: MAIN.bDO25
        toggle MAIN.bDO25
    Button (455,280 150x30), "DO 6", colour toggle: MAIN.bDO26
        toggle MAIN.bDO26
    Button (455,320 150x30), "DO 7", colour toggle: MAIN.bDO27
        toggle MAIN.bDO27
    Button (455,360 150x30), "DO 8", colour toggle: MAIN.bDO28
        toggle MAIN.bDO28
    Button (620,81 150x30), "DO 9", colour toggle: MAIN.bDO29
        toggle MAIN.bDO29
    Button (620,121 150x30), "DO 10", colour toggle: MAIN.bDO210
        toggle MAIN.bDO210
    Button (620,161 150x30), "DO 11", colour toggle: MAIN.bDO211
        toggle MAIN.bDO211
    Button (620,201 150x30), "DO 12", colour toggle: MAIN.bDO212
        toggle MAIN.bDO212
    Button (620,241 150x30), "DO 13", colour toggle: MAIN.bDO213
        toggle MAIN.bDO213
    Button (620,281 150x30), "DO 14", colour toggle: MAIN.bDO214
        toggle MAIN.bDO214
    Button (620,321 150x30), "DO 15", colour toggle: MAIN.bDO215
        toggle MAIN.bDO215
    Button (620,361 150x30), "DO 16", colour toggle: MAIN.bDO216
        toggle MAIN.bDO216
    Rectangle (850,81 150x30), "Analog 1"
    Rectangle (850,121 150x30), "Analog 2"
    Rectangle (850,201 150x30), "Analog 4"
    Rectangle (850,161 150x30), "Analog 3"
    Rectangle (850,281 150x30), "Analog 6"
    Rectangle (850,241 150x30), "Analog 5"
    Rectangle (850,321 150x30), "Analog 7"
    Rectangle (850,361 150x30), "Analog 8"
    Textfield (1170,81 150x30), "%2.8f", text variable: MAIN.lrGovernorGuideVaneOilPreesure
    Textfield (1170,121 150x30), "%2.8f", text variable: MAIN.lrGovernorBladeOilPressure
    Textfield (1170,161 150x30), "%2.8f", text variable: MAIN.lrExcitationVoltage
    Textfield (1170,201 150x30), "%2.8f", text variable: MAIN.lrExcitationCurrent
    Textfield (1170,241 150x30), "%2.8f", text variable: MAIN.lrSpiralCasePressure
    Textfield (1170,281 150x30), "%2.8f", text variable: MAIN.lrHeadCasePressure
    Textfield (1170,321 150x30), "%2.8f", text variable: MAIN.lrDraftT1CasePressure
    Textfield (1170,361 150x30), "%2.8f", text variable: MAIN.lrDraftT2CasePressure
    Rectangle (1170,41 150x30), "Current value"
    Rectangle (1330,81 150x30), "%s", text variable: MAIN.fbCal1.sDescription
    Rectangle (1330,121 150x30), "%s", text variable: MAIN.fbCal2.sDescription
    Rectangle (1330,201 150x30), "%s", text variable: MAIN.fbCal4.sDescription
    Rectangle (1330,161 150x30), "%s", text variable: MAIN.fbCal3.sDescription
    Rectangle (1330,281 150x30), "%s", text variable: MAIN.fbCal6.sDescription
    Rectangle (1330,241 150x30), "%s", text variable: MAIN.fbCal5.sDescription
    Rectangle (1330,321 150x30), "%s", text variable: MAIN.fbCal7.sDescription
    Rectangle (1330,361 150x30), "%s", text variable: MAIN.fbCal8.sDescription
    Textfield (1010,81 150x30), "%5d", text variable: MAIN.fbCal1.wRawIn
    Textfield (1010,121 150x30), "%5d", text variable: MAIN.fbCal2.wRawIn
    Textfield (1010,161 150x30), "%5d", text variable: MAIN.fbCal3.wRawIn
    Textfield (1010,201 150x30), "%5d", text variable: MAIN.fbCal4.wRawIn
    Textfield (1010,241 150x30), "%5d", text variable: MAIN.fbCal5.wRawIn
    Textfield (1010,281 150x30), "%5d", text variable: MAIN.fbCal6.wRawIn
    Textfield (1010,321 150x30), "%5d", text variable: MAIN.fbCal7.wRawIn
    Textfield (1010,361 150x30), "%5d", text variable: MAIN.fbCal8.wRawIn
    Rectangle (1010,41 150x30), "Raw value"
END_VISUALIZATION
